(* IEC 61131-3 sources: RL_MAR/experiments/comparison/llm4plc/results/gpt-4o_20260507_114630/20260507_121927, 2 files *)

(* ---- generated_code_iteration_0.st ---- *)
plaintext
START_ST
FUNCTION_BLOCK ParcelSortingSystem
VAR_INPUT
    ParcelSizeSensor : REAL; (* Sensor input for parcel size *)
    DestinationCodeSensor : INT; (* Destination code: 1=A, 2=B *)
END_VAR
VAR_OUTPUT
    ConveyorBeltMotor : BOOL; (* Output for conveyor belt motor: TRUE=On, FALSE=Off *)
    SortingGate1 : BOOL; (* Output for sorting gate 1: TRUE=Open, FALSE=Closed *)
    SortingGate2 : BOOL; (* Output for sorting gate 2: TRUE=Open, FALSE=Closed *)
END_VAR
VAR
    state : INT; (* Current state of the system *)
    prevState : INT; (* Previous state of the system *)
    LARGE_THRESHOLD : REAL := 50.0; (* Threshold for large parcel size *)
END_VAR

(* Initialize the system to STATE 0 *)
IF state = 0 THEN
    (* STATE 0: INITIALIZE *)
    ConveyorBeltMotor := FALSE; (* Turn off conveyor belt motor *)
    SortingGate1 := FALSE; (* Close sorting gate 1 *)
    SortingGate2 := FALSE; (* Close sorting gate 2 *)
    prevState := state; (* Store the current state as previous state *)
    state := 1; (* Transition to STATE 1 to begin processing parcels *)
END_IF

(* Check parcel validity and determine the next state *)
IF state = 1 THEN
    (* STATE 1: CHECK PARCEL VALIDITY *)
    ConveyorBeltMotor := TRUE; (* Turn on conveyor belt motor *)
    SortingGate1 := FALSE; (* Ensure sorting gate 1 is closed *)
    SortingGate2 := FALSE; (* Ensure sorting gate 2 is closed *)

    IF ParcelSizeSensor > LARGE_THRESHOLD THEN
        state := 2; (* Transition to STATE 2 for large parcels *)
    ELSIF (ParcelSizeSensor <= LARGE_THRESHOLD) AND (DestinationCodeSensor = 1) THEN
        state := 3; (* Transition to STATE 3 for small parcels to location A *)
    ELSIF (ParcelSizeSensor <= LARGE_THRESHOLD) AND (DestinationCodeSensor = 2) THEN
        state := 4; (* Transition to STATE 4 for small parcels to location B *)
    ELSIF (ParcelSizeSensor <= 0) OR (DestinationCodeSensor NOT IN [1, 2]) THEN
        state := 5; (* Transition to STATE 5 for invalid inputs *)
    END_IF
END_IF

(* Handle large parcels *)
IF state = 2 THEN
    (* STATE 2: SORT LARGE PARCELS *)
    ConveyorBeltMotor := TRUE; (* Keep the conveyor belt running *)
    SortingGate1 := TRUE; (* Open sorting gate 1 *)
    SortingGate2 := FALSE; (* Ensure sorting gate 2 is closed *)
    prevState := state; (* Store the current state as previous state *)
    state := 0; (* Transition back to STATE 0 after sorting operation *)
END_IF

(* Handle small parcels destined for location A *)
IF state = 3 THEN
    (* STATE 3: SORT SMALL PARCELS TO LOCATION A *)
    ConveyorBeltMotor := TRUE; (* Keep the conveyor belt running *)
    SortingGate1 := FALSE; (* Ensure sorting gate 1 is closed *)
    SortingGate2 := TRUE; (* Open sorting gate 2 *)
    prevState := state; (* Store the current state as previous state *)
    state := 0; (* Transition back to STATE 0 after sorting operation *)
END_IF

(* Handle small parcels destined for location B *)
IF state = 4 THEN
    (* STATE 4: SORT SMALL PARCELS TO LOCATION B *)
    ConveyorBeltMotor := TRUE; (* Keep the conveyor belt running *)
    SortingGate1 := FALSE; (* Ensure sorting gate 1 is closed *)
    SortingGate2 := FALSE; (* Ensure sorting gate 2 is closed *)
    prevState := state; (* Store the current state as previous state *)
    state := 0; (* Transition back to STATE 0 after parcel moves past conveyor belt *)
END_IF

(* Handle invalid inputs *)
IF state = 5 THEN
    (* STATE 5: ERROR HANDLING *)
    ConveyorBeltMotor := FALSE; (* Stop the conveyor belt *)
    SortingGate1 := FALSE; (* Close sorting gate 1 *)
    SortingGate2 := FALSE; (* Close sorting gate 2 *)
    prevState := state; (* Store the current state as previous state *)
    state := 0; (* Transition back to STATE 0 after error handling *)
END_IF

END_FUNCTION_BLOCK
END_ST

(* ---- generated_code_iteration_1.st ---- *)
START_REASON
The validation feedback indicates that the CODESYS compiler validation failed due to the incorrect use of `NOT` in the expression `(DestinationCodeSensor NOT IN [1, 2])`. In Structured Text (ST), the `NOT` operator is used for logical negation, and the syntax `NOT IN` is not valid. Instead, the expression should be corrected to use proper logical negation and comparison operators to achieve the intended functionality.

The error occurred because the syntax for checking if a value is not in a set was incorrectly implemented. The correct approach is to use logical comparisons explicitly to check if the value does not match any of the specified values.

To fix this issue, I will replace `(DestinationCodeSensor NOT IN [1, 2])` with an equivalent logical comparison that checks if `DestinationCodeSensor` is neither `1` nor `2`.
END_REASON

START_ST
FUNCTION_BLOCK ParcelSortingSystem
VAR_INPUT
    ParcelSizeSensor : REAL; (* Sensor input for parcel size *)
    DestinationCodeSensor : INT; (* Destination code: 1=A, 2=B *)
END_VAR
VAR_OUTPUT
    ConveyorBeltMotor : BOOL; (* Output for conveyor belt motor: TRUE=On, FALSE=Off *)
    SortingGate1 : BOOL; (* Output for sorting gate 1: TRUE=Open, FALSE=Closed *)
    SortingGate2 : BOOL; (* Output for sorting gate 2: TRUE=Open, FALSE=Closed *)
END_VAR
VAR
    state : INT; (* Current state of the system *)
    prevState : INT; (* Previous state of the system *)
    LARGE_THRESHOLD : REAL := 50.0; (* Threshold for large parcel size *)
END_VAR

(* Initialize the system to STATE 0 *)
IF state = 0 THEN
    (* STATE 0: INITIALIZE *)
    ConveyorBeltMotor := FALSE; (* Turn off conveyor belt motor *)
    SortingGate1 := FALSE; (* Close sorting gate 1 *)
    SortingGate2 := FALSE; (* Close sorting gate 2 *)
    prevState := state; (* Store the current state as previous state *)
    state := 1; (* Transition to STATE 1 to begin processing parcels *)
END_IF

(* Check parcel validity and determine the next state *)
IF state = 1 THEN
    (* STATE 1: CHECK PARCEL VALIDITY *)
    ConveyorBeltMotor := TRUE; (* Turn on conveyor belt motor *)
    SortingGate1 := FALSE; (* Ensure sorting gate 1 is closed *)
    SortingGate2 := FALSE; (* Ensure sorting gate 2 is closed *)

    IF ParcelSizeSensor > LARGE_THRESHOLD THEN
        state := 2; (* Transition to STATE 2 for large parcels *)
    ELSIF (ParcelSizeSensor <= LARGE_THRESHOLD) AND (DestinationCodeSensor = 1) THEN
        state := 3; (* Transition to STATE 3 for small parcels to location A *)
    ELSIF (ParcelSizeSensor <= LARGE_THRESHOLD) AND (DestinationCodeSensor = 2) THEN
        state := 4; (* Transition to STATE 4 for small parcels to location B *)
    ELSIF (ParcelSizeSensor <= 0) OR ((DestinationCodeSensor <> 1) AND (DestinationCodeSensor <> 2)) THEN
        state := 5; (* Transition to STATE 5 for invalid inputs *)
    END_IF
END_IF

(* Handle large parcels *)
IF state = 2 THEN
    (* STATE 2: SORT LARGE PARCELS *)
    ConveyorBeltMotor := TRUE; (* Keep the conveyor belt running *)
    SortingGate1 := TRUE; (* Open sorting gate 1 *)
    SortingGate2 := FALSE; (* Ensure sorting gate 2 is closed *)
    prevState := state; (* Store the current state as previous state *)
    state := 0; (* Transition back to STATE 0 after sorting operation *)
END_IF

(* Handle small parcels destined for location A *)
IF state = 3 THEN
    (* STATE 3: SORT SMALL PARCELS TO LOCATION A *)
    ConveyorBeltMotor := TRUE; (* Keep the conveyor belt running *)
    SortingGate1 := FALSE; (* Ensure sorting gate 1 is closed *)
    SortingGate2 := TRUE; (* Open sorting gate 2 *)
    prevState := state; (* Store the current state as previous state *)
    state := 0; (* Transition back to STATE 0 after sorting operation *)
END_IF

(* Handle small parcels destined for location B *)
IF state = 4 THEN
    (* STATE 4: SORT SMALL PARCELS TO LOCATION B *)
    ConveyorBeltMotor := TRUE; (* Keep the conveyor belt running *)
    SortingGate1 := FALSE; (* Ensure sorting gate 1 is closed *)
    SortingGate2 := FALSE; (* Ensure sorting gate 2 is closed *)
    prevState := state; (* Store the current state as previous state *)
    state := 0; (* Transition back to STATE 0 after parcel moves past conveyor belt *)
END_IF

(* Handle invalid inputs *)
IF state = 5 THEN
    (* STATE 5: ERROR HANDLING *)
    ConveyorBeltMotor := FALSE; (* Stop the conveyor belt *)
    SortingGate1 := FALSE; (* Close sorting gate 1 *)
    SortingGate2 := FALSE; (* Close sorting gate 2 *)
    prevState := state; (* Store the current state as previous state *)
    state := 0; (* Transition back to STATE 0 after error handling *)
END_IF

END_FUNCTION_BLOCK
END_ST
